(* PLC project KinIn_v3.project, CODESYS CODESYS V3.5 SP19 *)
(* stored: creationDateTime 2025-01-20T16:27:34.7649156, modificationDateTime 2025-01-20T16:17:39.6822999 *)

FUNCTION_BLOCK norm
  VAR_INPUT
    {attribute 'variable_length_array_original_scope' := 'Inout'}
    {attribute 'variable_length_array' := 'ARRAY[*] OF REAL'}
    {attribute 'Dimensions' := '1'}
    vector : POINTER TO REAL;  (* vector *)
  END_VAR
  VAR_OUTPUT
    normValue : REAL;
  END_VAR
  VAR
    i : DINT;
  END_VAR

            //This get the norm of the vector
normValue:=0;
FOR i:=1 TO UPPER_BOUND(vector,1) DO
	normValue:=normValue+vector[i]*vector[i];
END_FOR
normValue:=SQRT(normValue);

          
END_FUNCTION_BLOCK
